TYPE ST_PyAdsQuit:
  STRUCT
    bDone : BOOL;
    bError: BOOL;
  END_STRUCT
END_TYPE

(* stored: Version 1.1.0.1, ProductVersion 3.1.4024.2
   DUT ST_PyAdsQuit: Id {57ee0c64-6e94-48bc-adf5-6e0f80c38c1d} *)
